FUNCTION_BLOCK ModuleBase
VAR
	fbAxis			:		ARRAY[1..mcGlobal.cMaxNoOfAxis] OF AxisBase[
															(AxisName		:=	'Axis1',
															nPtpPoints		:=	5,
															iProcessHandler	:=	0,
															iTorqueLimiting	:=	0,
															iPosCamLookup	:=	0,
															iVeloCamLookup	:=	0,
															iPtpCamLookup	:=	0),
															(AxisName		:=	'Axis2',
															nPtpPoints		:=	5,
															iProcessHandler	:=	0,
															iTorqueLimiting	:=	0,
															iPosCamLookup	:=	0,
															iVeloCamLookup	:=	0,
															iPtpCamLookup	:=	0),
															(AxisName		:=	'Axis3',
															nPtpPoints		:=	5,
															iProcessHandler	:=	0,
															iTorqueLimiting	:=	0,
															iPosCamLookup	:=	0,
															iVeloCamLookup	:=	0,
															iPtpCamLookup	:=	0),
															(AxisName		:=	'Axis4',
															nPtpPoints		:=	5,
															iProcessHandler	:=	0,
															iTorqueLimiting	:=	0,
															iPosCamLookup	:=	0,
															iVeloCamLookup	:=	0,
															iPtpCamLookup	:=	0),
															(AxisName		:=	'Axis5',
															nPtpPoints		:=	5,
															iProcessHandler	:=	0,
															iTorqueLimiting	:=	0,
															iPosCamLookup	:=	0,
															iVeloCamLookup	:=	0,
															iPtpCamLookup	:=	0),
															(AxisName		:=	'Axis6',
															nPtpPoints		:=	5,
															iProcessHandler	:=	0,
															iTorqueLimiting	:=	0,
															iPosCamLookup	:=	0,
															iVeloCamLookup	:=	0,
															iPtpCamLookup	:=	0),
															(AxisName		:=	'Axis7',
															nPtpPoints		:=	5,
															iProcessHandler	:=	0,
															iTorqueLimiting	:=	0,
															iPosCamLookup	:=	0,
															iVeloCamLookup	:=	0,
															iPtpCamLookup	:=	0),
															(AxisName		:=	'Axis8',
															nPtpPoints		:=	5,
															iProcessHandler	:=	0,
															iTorqueLimiting	:=	0,
															iPosCamLookup	:=	0,
															iVeloCamLookup	:=	0,
															iPtpCamLookup	:=	0)
															];
	iCount				:		INT;
END_VAR

VAR_INPUT
	intNoOfAxis			:		INT;
END_VAR

FOR iCount := 1 TO intNoOfAxis DO
	fbAxis[iCount].A_Cyclic();
END_FOR

END_FUNCTION_BLOCK

(* stored: Version 1.1.0.1, ProductVersion 3.1.4024.6
   POU ModuleBase: Id {de1993d4-1e1b-43b1-8448-164441f29cf7}, SpecialFunc None *)
